// TwinCAT 3 PLC project PLC1
// ProgramVersion: 3.1.4023.0
// libraries:
//   Tc2_ControllerToolbox, * (Beckhoff Automation GmbH)
//   Tc2_SPA, * (Beckhoff Automation GmbH)
//   Tc2_Standard, * (Beckhoff Automation GmbH)
//   Tc2_System, * (Beckhoff Automation GmbH)
//   Tc3_Module, * (Beckhoff Automation GmbH)
//   VisuDialogs, * (System)
//   Tc2_Math,3.3.1.0,Beckhoff Automation GmbH
// project tree:
//   DUTs/ ST_AdvancedTanks.TcDUT, ST_Tanks.TcDUT
//   / GlobalTextList.TcGTLO, PlcTask.TcTTO, Visualization Manager.TcVMO (not stored), VISU_TASK.TcTTO
//   POUs/ FB_Pulse.TcPOU, Func_example.TcPOU, F_CtoF.TcPOU, IF_Statement.TcPOU, MAIN.TcPOU, Func_block_example.TcPOU, Structs_example.TcPOU
//   VISUs/ Viz1.TcVIS
// real-time tasks:
//   TASK PlcTask: cycle T#10ms, priority 20, ADS port 350
//   TASK VISU_TASK: cycle T#200000us, priority 30, ADS port 351

CONFIGURATION PLC1
    RESOURCE PLC ON TwinCAT3
        TASK PlcTask(INTERVAL := T#10ms, PRIORITY := 20);
        TASK VISU_TASK(INTERVAL := T#200000us, PRIORITY := 30);
        PROGRAM MAIN WITH PlcTask : MAIN;
        PROGRAM Func_example WITH PlcTask : Func_example;
        PROGRAM Structs_example WITH PlcTask : Structs_example;
        PROGRAM Func_block_example WITH PlcTask : Func_block_example;
        PROGRAM IF_Statement WITH PlcTask : IF_Statement;
        PROGRAM VisuElems_Visu_Prg WITH VISU_TASK : VisuElems.Visu_Prg;
    END_RESOURCE
END_CONFIGURATION

// ---- DUTs/ST_AdvancedTanks.TcDUT
TYPE ST_AdvancedTanks EXTENDS ST_Tanks :
STRUCT
	rPressure : REAL;
END_STRUCT
END_TYPE

// ---- DUTs/ST_Tanks.TcDUT
TYPE ST_Tanks :
STRUCT
	iLevel : INT;
	rTemp : REAL;
	xStatus : BOOL := TRUE;
	sDescription : STRING;
	
END_STRUCT
END_TYPE

// ---- POUs/MAIN.TcPOU
PROGRAM MAIN
VAR
	//Inputs
	iNumber : INT;
	bSwitch1 : BOOL;
	bSwitch2 : BOOL;
	bSwitch3 : BOOL;
	bSwitch4 : BOOL;
	//Outputs
	bLight1 : BOOL;
	bLight2 : BOOL;
	bLight3 : BOOL;
	bLight4 : BOOL;
	aLights : ARRAY[1..4] OF BOOL;
	i : INT;
	aCounter : ARRAY[1..10] OF INT:= [1,2,3,4,5,6,7,8,9,10];
	iCounterDisp : INT;
	index : INT := 0;
	iStep: INT;	
END_VAR

FOR i := 1 TO 4 DO
	aLights[i] := FALSE;
END_FOR

// ARRAY Example
CASE iNumber OF
	0..8000:
		aLights[1] := TRUE;
	8001..16000:
		aLights[2] := TRUE;
	16001..24000:
		aLights[3] := TRUE;
	ELSE
		aLights[4] := TRUE;
END_CASE

Structs_example();

(*
// CASE Example
bLight1 := bLight2 := bLight3 := bLight4 := FALSE;
CASE iNumber OF
	0..8000:
		bLight1 := TRUE;
	8001..16000:
		bLight2 := TRUE;
	16001..24000:
		bLight3 := TRUE;
	ELSE
		bLight4 := TRUE;
END_CASE
*)



(*
index := index + 1;
iCounterDisp := aCounter[index];

IF index > 10 THEN
	index := 0;
END_IF

IF_Statement();
*)

END_PROGRAM

// ---- POUs/Structs_example.TcPOU
PROGRAM Structs_example
VAR
	stTank1 : ST_Tanks;
	stTank2 : ST_Tanks;	
	xSetTemps : BOOL;
	stTank3 : ST_AdvancedTanks;  // Structure that extends ST_Tanks structure.  Inherits fields from ST_Tanks	
END_VAR

IF xSetTemps = TRUE THEN
	stTank1.rTemp := 100.0;
	stTank2.rTemp := 50.0;
END_IF

END_PROGRAM

// ---- POUs/Func_example.TcPOU
PROGRAM Func_example
VAR
	iMyInt : INT;
	uMyInt : INT;
	TmpC : LREAL;
	TmpF : LREAL;
END_VAR

iMyInt := UINT_TO_INT(uMyInt);

TmpF := F_CtoF(TmpC);

END_PROGRAM

// ---- POUs/F_CtoF.TcPOU
FUNCTION F_CtoF : LREAL
VAR_INPUT
	lrTempInC : LREAL;
END_VAR
VAR
END_VAR

F_CtoF := lrTempInC * (9.0/5.0) + 32.0;

END_FUNCTION

// ---- POUs/Func_block_example.TcPOU
PROGRAM Func_block_example
VAR
	myCounter : CTU;
	bCountUp: BOOL;
	bReset: BOOL;
	bCountDone: BOOL;
	myPulse : FB_Pulse;
	myPulse2 : FB_Pulse;
END_VAR

myCounter(
	CU:= bCountUp,
	RESET := bReset,
	PV:= 5, 
	Q=>bCountDone , 
	CV=> );
	
	
myPulse(bEnable:= , tTimeOn:= T#1S, tTimeOff:= T#500MS, bPulse=> );

myPulse2();

END_PROGRAM

// ---- POUs/FB_Pulse.TcPOU
FUNCTION_BLOCK FB_Pulse
VAR_INPUT
	bEnable : BOOL;
	tTimeOn : TIME;
	tTimeOff : TIME;
END_VAR
VAR_OUTPUT
	bPulse : BOOL;
END_VAR
VAR
	tmr1 : TON;
	tmr2 : TOF;
	IN: INT;
END_VAR

tmr1(IN:= bEnable AND NOT tmr2.Q, PT:= tTimeOff, Q=> , ET=> );
tmr2(IN:= tmr1.Q, PT:= tTimeOn, Q=> bPulse, ET=> );

END_FUNCTION_BLOCK

// ---- POUs/IF_Statement.TcPOU
PROGRAM IF_Statement

VAR
	//Inputs
	iNumber : INT;
	bSwitch1 : BOOL;
	bSwitch2 : BOOL;
	bSwitch3 : BOOL;
	bSwitch4 : BOOL;
	//Outputs
	bLight1 : BOOL;
	bLight2 : BOOL;
	bLight3 : BOOL;
	bLight4 : BOOL;
END_VAR

// IF statement example
bLight1 := bLight2 := bLight3 := bLight4 := FALSE; 

IF iNumber >= 0 AND iNumber <= 8000 THEN
	bLight1 := TRUE;	
ELSIF iNumber > 8000 AND iNumber <= 16000 THEN
	bLight2 := TRUE;	
ELSIF iNumber > 16000 AND iNumber <= 24000 THEN
	bLight3 := TRUE;	
ELSE 
	bLight4 := TRUE;		
END_IF

END_PROGRAM

// ---- GlobalTextList.TcGTLO
TEXTLIST GlobalTextList
  475 = '%i'
  341 = '%s'
  234 = '1'
  38 = '2'
  410 = '3'
  690 = '4'
  207 = 'Display'
  666 = 'Disply'
  824 = 'Input'
END_TEXTLIST

// ---- VISUs/Viz1.TcVIS
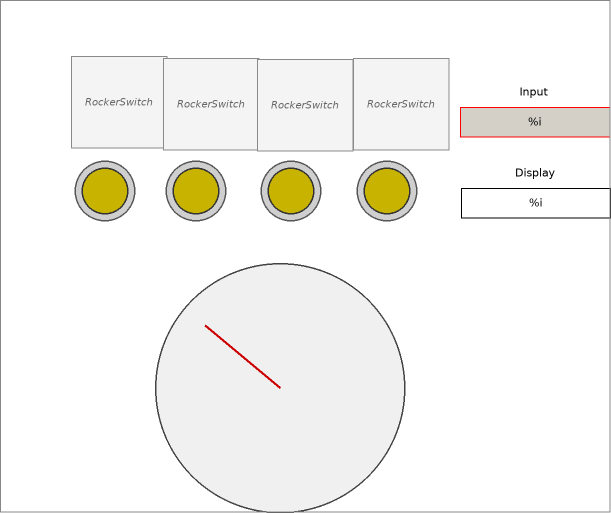
VISUALIZATION Viz1  // 611x513
    Lamp1 (70,156 70x70), variable: IF_Statement.bLight1, style: Lamp-Lamp1-Yellow
    Lamp1 (161,156 70x70), variable: IF_Statement.bLight2, style: Lamp-Lamp1-Yellow
    Lamp1 (256,156 70x70), variable: IF_Statement.bLight3, style: Lamp-Lamp1-Yellow
    Lamp1 (352,156 70x70), variable: IF_Statement.bLight4, style: Lamp-Lamp1-Yellow
    Rectangle (460,107 150x30), "%i", text variable: IF_Statement.iNumber
        OnMouseDown: write the text variable via Default
    Rectangle (461,188 150x30), "%i", text variable: MAIN.iCounterDisp
    Label (459,77 150x30), "Input"
    Label (460,158 150x30), "Display"
    RockerSwitch (71,56 96x92), variable: IF_Statement.bSwitch1, behaviour: TOGGLE, style: Switch-RockerSwitch-Gray
    RockerSwitch (163,58 96x92), variable: IF_Statement.bSwitch2, behaviour: TOGGLE, style: Switch-RockerSwitch-Gray
    RockerSwitch (257,59 96x92), variable: IF_Statement.bSwitch3, behaviour: TOGGLE, style: Switch-RockerSwitch-Gray
    RockerSwitch (353,58 96x92), variable: IF_Statement.bSwitch4, behaviour: TOGGLE, style: Switch-RockerSwitch-Gray
    Meter360 (155,263 250x250), value: IF_Statement.iNumber, style: Meter-Meter360-Gray, scale format: %.1f, scale 0..32000
END_VISUALIZATION
